Staubli VAL3: getTool.pgx

public program getTool(tool& x_tTool[] (dimensions=1), num x_nIndex (dimensions=1))
begin
  // get the tool
  x_tTool=tData[x_nIndex].tcp
end
